TYPE E_CylinderPosition :
(
	eCylinderPosition_unknown := 0,
	eCylinderPosition_hp,
	eCylinderPosition_mp,
	eCylinderPosition_wp
);
END_TYPE

(* stored: Version 1.1.0.1, ProductVersion 3.1.4022.9
   DUT E_CylinderPosition: Id {0f0b6b01-9177-41ef-af84-4450136fa4db} *)
